FUNCTION_BLOCK DAerationLogic (* Composite Function Block Type *)
  (* Standard: 61499-2 *)
  (* Version 0.0, 10/24/2023, SESA685388, Schneider Electric, template *)
  PACKAGE SE.Nereda;
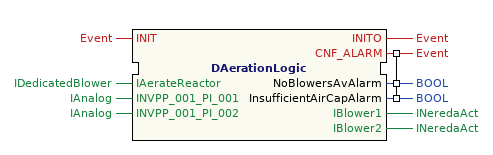
  EVENT_INPUT
    INIT; (* Initialization Request *)
  END_EVENT
  EVENT_OUTPUT
    INITO; (* Initialization Confirm *)
    CNF_ALARM WITH NoBlowersAvAlarm, InsufficientAirCapAlarm; (* Execution Confirmation *)
  END_EVENT
  VAR_OUTPUT
    NoBlowersAvAlarm : BOOL; (* Output event qualifier *)
    InsufficientAirCapAlarm : BOOL; (* Output event qualifier *)
  END_VAR
  SOCKETS
    IAerateReactor : IDedicatedBlower;
    INVPP_001_PI_001 : IAnalog;
    INVPP_001_PI_002 : IAnalog;
  END_SOCKETS
  PLUGS
    IBlower1 : INeredaAct;
    IBlower2 : INeredaAct;
  END_PLUGS
  (* 01 - FUNCTIONNAL INPUT INTERFACE *)
  (* 00 - INITIALIZATION *)
  (* 05 - LOGIC *)
  (* 06 - HMI INTERFACE *)
  (* CommandLogic *)
  (* 02 - FUNCTIONNAL OUTPUT INTERFACE *)
  (* Aeration Capacity Sp *)
  (* Blowers State *)
  FBS
    BlowersFbReady : AND_88A3DD8EC65DD11C; {SET_ATTRIBUTE(Configuration.GenericFBType.InterfaceParams, Runtime.Standard#CNT:=2;OUT:BOOL)}
    CommandLogic : DAerationLogicBasic;
    Blower1Cmd_Smooth : boolValueChanged;
    Blower2Cmd_Smooth : boolValueChanged;
    IThis : DAerationLogic_HMI(QI := TRUE);
    BlowersFbStopped : AND_88A3DD8EC65DD11C; {SET_ATTRIBUTE(Configuration.GenericFBType.InterfaceParams, Runtime.Standard#CNT:=2;OUT:BOOL)}
    BlowersFbRunning : OR_88A3DD8EC65DD11C; {SET_ATTRIBUTE(Configuration.GenericFBType.InterfaceParams, Runtime.Standard#CNT:=2;OUT:BOOL)}
    CapacityCalculated : NeredaCapacitySpToDBlowersSp;
    TowBlowersRunning : AND_88A3DD8EC65DD11C; {SET_ATTRIBUTE(Configuration.GenericFBType.InterfaceParams, Runtime.Standard#CNT:=2;OUT:BOOL)}
    NVPP_001_PI_001_Status : decodeStatus; {SET_ATTRIBUTE(Configuration.Component.HideUnusedPorts, )}
    NVPP_001_PI_002_Status : decodeStatus; {SET_ATTRIBUTE(Configuration.Component.HideUnusedPorts, )}
    Blower1Cmd : BOOL2INT;
    Blower2Cmd : BOOL2INT;
    AlarmsManager : CheckOneBlReady;
  END_FBS
  EVENT_CONNECTIONS
    BlowersFbRunning.CNF TO BlowersFbStopped.REQ;
    BlowersFbStopped.CNF TO TowBlowersRunning.REQ;
    INVPP_001_PI_001.REQ_STATUS TO NVPP_001_PI_001_Status.REQ;
    INVPP_001_PI_002.REQ_STATUS TO NVPP_001_PI_002_Status.REQ;
    INIT TO IThis.73B62E902A5807A1;
    IThis.F68012C9A80C276B TO IThis.559778F4ADF98A31;
    IThis.3F1A2A449466611E TO IThis.1EFA35ABAB87DA3F;
    IThis.F68012C9A80C276B TO INITO;
    IThis.B2C582118AFFEE3D TO IThis.354838261F992C4A;
    IAerateReactor.START_BLOWER TO CommandLogic.D2C11A8772DD75BE;
    IAerateReactor.FLOW_SP_BLOWER TO CapacityCalculated.D0388ADF8D5604CA;
    IAerateReactor.FLOW_SP_BLOWER TO IThis.D425E5A096E0D21E;
    TowBlowersRunning.CNF TO IAerateReactor.FB_BLOWER;
    AlarmsManager.F3042427BFA42A43 TO IAerateReactor.FB_BLOWER_AVAILABLE;
    NVPP_001_PI_001_Status.CNF TO CommandLogic.1B0353354B77DB6A;
    NVPP_001_PI_002_Status.CNF TO CommandLogic.1B0353354B77DB6A;
    CommandLogic.F0F26EFFA0ABF35A TO IThis.D9F2C8BAFB22D330;
    IBlower1.2DA8AEC15204E92D TO IThis.4600AA800ADCB9DD;
    IBlower2.2DA8AEC15204E92D TO IThis.4600AA800ADCB9DD;
    CommandLogic.3AB27F52460EDDB2 TO IThis.3A50EC6A27D39101;
    CapacityCalculated.CNF TO IThis.3A50EC6A27D39101;
    IThis.3F1A2A449466611E TO CommandLogic.979DF616CA3CB55A;
    IThis.3F1A2A449466611E TO CapacityCalculated.D0388ADF8D5604CA;
    IThis.B2C582118AFFEE3D TO CapacityCalculated.D0388ADF8D5604CA;
    IBlower1.9CD053F8408797ED TO BlowersFbRunning.REQ;
    IBlower2.9CD053F8408797ED TO BlowersFbRunning.REQ;
    IBlower1.CC753684FA882790 TO BlowersFbReady.REQ;
    IBlower2.CC753684FA882790 TO BlowersFbReady.REQ;
    AlarmsManager.F3042427BFA42A43 TO CommandLogic.C2CA1F9B44AEDC08;
    TowBlowersRunning.CNF TO CapacityCalculated.D0388ADF8D5604CA;
    CommandLogic.1ADA5B269032EF11 TO CapacityCalculated.D0388ADF8D5604CA;
    CapacityCalculated.CNF TO CommandLogic.BF57157246C0E97B;
    IBlower1.F846995A4121D865 TO CommandLogic.13BA3066C47C3D65;
    IBlower2.F846995A4121D865 TO CommandLogic.13BA3066C47C3D65;
    TowBlowersRunning.CNF TO CommandLogic.13BA3066C47C3D65;
    IBlower1.2DA8AEC15204E92D TO CommandLogic.349546B416B30E3C;
    IBlower2.2DA8AEC15204E92D TO CommandLogic.349546B416B30E3C;
    CommandLogic.B804F7AE49CF3E15 TO Blower1Cmd_Smooth.REQ;
    CommandLogic.B804F7AE49CF3E15 TO Blower2Cmd_Smooth.REQ;
    CommandLogic.3AB27F52460EDDB2 TO IBlower1.1E00729184986247;
    CommandLogic.3AB27F52460EDDB2 TO IBlower2.1E00729184986247;
    Blower1Cmd_Smooth.CHD TO Blower1Cmd.DD5870AA881150BB;
    Blower2Cmd_Smooth.CHD TO Blower2Cmd.DD5870AA881150BB;
    Blower1Cmd.6FC99A5BD1C38561 TO IBlower1.0F1CDF9A9B4A227A;
    Blower2Cmd.6FC99A5BD1C38561 TO IBlower2.0F1CDF9A9B4A227A;
    AlarmsManager.F3042427BFA42A43 TO CNF_ALARM;
    BlowersFbReady.CNF TO AlarmsManager.2E84B14BD871A818;
  END_CONNECTIONS
  DATA_CONNECTIONS
    INVPP_001_PI_001.Status TO NVPP_001_PI_001_Status.Status;
    INVPP_001_PI_002.Status TO NVPP_001_PI_002_Status.Status;
    IThis.AA0BF853026C240A TO IThis.6AF7DF1BED298D82;
    IThis.1A24AFB83170123C TO IThis.B0E59345C5AABE21;
    IThis.A8DDE26075A11F35 TO IThis.6D59C4836DAB0D3F;
    IThis.E5E878DDA85BBBF4 TO IThis.8B0D715E2C883E41;
    IAerateReactor.StartBlower TO CommandLogic.B2CC9DAB470B3A98;
    IAerateReactor.FlowSPBlower TO CommandLogic.09FC2180130EA7A8;
    IAerateReactor.FlowSPBlower TO CapacityCalculated.Setpoint;
    IAerateReactor.FlowSPBlower TO IThis.177565698FAA90E6;
    BlowersFbRunning.OUT TO IAerateReactor.FBStart;
    BlowersFbStopped.OUT TO IAerateReactor.FBStop;
    BlowersFbReady.OUT TO IAerateReactor.FBBlowersAbailable;
    NVPP_001_PI_001_Status.HiHiAlarm TO CommandLogic.3701C14F32674847;
    NVPP_001_PI_002_Status.HiHiAlarm TO CommandLogic.70B7D0989DE93DE6;
    CommandLogic.C09FEE22885584F4 TO IThis.B5F0A8EA6DDEEEEC;
    IBlower1.C7F638DBF6B860D2 TO IThis.1586E1E54C495A97;
    IBlower2.C7F638DBF6B860D2 TO IThis.56B8F4A164C3C697;
    IBlower1.10624535249F94F3 TO IThis.BB442219069ED8C4;
    IBlower2.10624535249F94F3 TO IThis.72677416375D933C;
    CommandLogic.EA9B07A85C385EDE TO IThis.7FB040E91AF01FE0;
    IThis.AA0BF853026C240A TO CommandLogic.A08DC9D6B6A9A9C5;
    IThis.AA0BF853026C240A TO CapacityCalculated.C_MAX;
    IThis.1A24AFB83170123C TO CommandLogic.BB0AA5D7C20FC6DC;
    IThis.A8DDE26075A11F35 TO CommandLogic.82E6F957CA34CE22;
    IThis.E5E878DDA85BBBF4 TO CapacityCalculated.160780B0FA04E6CC;
    IBlower1.B762734C094A7162 TO BlowersFbRunning.IN1;
    IBlower2.B762734C094A7162 TO BlowersFbRunning.IN2;
    IBlower1.D83B5BDEFA4D797C TO BlowersFbStopped.IN1;
    IBlower2.D83B5BDEFA4D797C TO BlowersFbStopped.IN2;
    IBlower1.B762734C094A7162 TO TowBlowersRunning.IN1;
    IBlower2.B762734C094A7162 TO TowBlowersRunning.IN2;
    TowBlowersRunning.OUT TO CapacityCalculated.Fb2BLRun;
    IBlower1.8A8A07EFCDA1443C TO BlowersFbReady.IN1;
    IBlower2.8A8A07EFCDA1443C TO BlowersFbReady.IN2;
    CommandLogic.86F036F9D0AC2083 TO CapacityCalculated.2DED152C27F3FC41;
    CapacityCalculated.SpeedBlower TO CommandLogic.DA5588204184617D;
    CommandLogic.6F30DD159F832B4D TO Blower1Cmd_Smooth.Input;
    CommandLogic.50D97D2FBAA8D1BB TO Blower2Cmd_Smooth.Input;
    CommandLogic.EA9B07A85C385EDE TO IBlower1.1BC103921BBFDA0B;
    CommandLogic.EA9B07A85C385EDE TO IBlower2.1BC103921BBFDA0B;
    Blower1Cmd_Smooth.Output TO Blower1Cmd.4573FC8F228EB71D;
    Blower2Cmd_Smooth.Output TO Blower2Cmd.4573FC8F228EB71D;
    Blower1Cmd.A6DEF5F9C27C1848 TO IBlower1.710D7FC54EE3F35A;
    IBlower1.790C5C3BA88E0AF5 TO CommandLogic.577CA07BFE5247BC;
    IBlower1.B762734C094A7162 TO CommandLogic.AF84CB02D2B46EA7;
    IBlower1.D83B5BDEFA4D797C TO CommandLogic.CF3BA6B848432326;
    IBlower1.8A8A07EFCDA1443C TO CommandLogic.0D2984DD8432BDE4;
    IBlower1.C7F638DBF6B860D2 TO CommandLogic.1198AC713518BF96;
    IBlower1.10624535249F94F3 TO CommandLogic.4207E8B5F773F643;
    Blower2Cmd.A6DEF5F9C27C1848 TO IBlower2.710D7FC54EE3F35A;
    IBlower2.D83B5BDEFA4D797C TO CommandLogic.B3E98BF14349172D;
    IBlower2.B762734C094A7162 TO CommandLogic.46433B3BDDEA2E25;
    IBlower2.790C5C3BA88E0AF5 TO CommandLogic.274CF35B495F03D7;
    IBlower2.8A8A07EFCDA1443C TO CommandLogic.266E7B658D2D8018;
    IBlower2.C7F638DBF6B860D2 TO CommandLogic.0E91FA9948C61E3C;
    IBlower2.10624535249F94F3 TO CommandLogic.83358589D0E93502;
    AlarmsManager.EE3ED52C74CC0874 TO InsufficientAirCapAlarm;
    AlarmsManager.4E7661CAE00B8F7F TO NoBlowersAvAlarm;
    IBlower1.8A8A07EFCDA1443C TO AlarmsManager.B6DDA2768C4989D9;
    IBlower2.8A8A07EFCDA1443C TO AlarmsManager.2DAF5142D84D4216;
  END_CONNECTIONS
END_FUNCTION_BLOCK
